FUNCTION_BLOCK ZERO_POS (* Set position value to 0,0,0 *)
  (* Standard: 61499-2 *)
  (* Version 1.0, 14-04-2012, GASR, Universidade do Estado de Santa Catarina *)
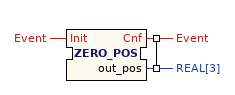
  EVENT_INPUT
    Init;
  END_EVENT
  EVENT_OUTPUT
    Cnf WITH out_pos;
  END_EVENT
  VAR_OUTPUT
    out_pos : ARRAY [0..2] OF REAL;
  END_VAR
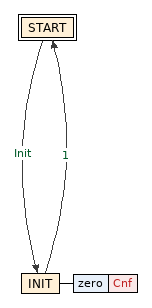
  EC_STATES
    START;
    INIT : zero -> Cnf;
  END_STATES
  EC_TRANSITIONS
    START TO INIT := Init;
    INIT TO START := 1;
  END_TRANSITIONS
  ALGORITHM zero IN Lua:
out_pos[1] = 0
out_pos[2] = 0
out_pos[3] = 0
  END_ALGORITHM
END_FUNCTION_BLOCK
